// TIA Portal V16 export
// export: Created 2024-12-03T15:41:45.3011474Z, ExportSetting WithReadOnly, DisplayName Totally Integrated Automation Portal, DisplayVersion V16 Update 6, DisplayName TIA Portal Version Control Interface, DisplayVersion V16 Update 2, DisplayName TIA Portal Openness, DisplayVersion V16 Update 6, DisplayName TIA Portal Teamcenter Gateway, DisplayVersion V16, DisplayName SINAMICS Startdrive Advanced, DisplayVersion V16 Update 5, DisplayName SINAMICS Startdrive G130, G150, S120, S150, SINAMICS MV, S210, DisplayVersion V16 Update 5, DisplayName SINAMICS Startdrive G110M, G120, G120C, G120D, G120P, G115D, DisplayVersion V16 Update 5, DisplayName STEP 7 Professional, DisplayVersion V16 Update 6, DisplayName STEP 7 Safety, DisplayVersion V16, DisplayName WinCC Advanced / Unified PC, DisplayVersion V16 Update 6
TYPE "COGNEX_DATAMAN_LOGIC_UDT"
TITLE = SICK Lector/CLV6xx data type
// This data type includes arguments and results using by the SICK_Lector_CLV6xx_PNDP function block.
// stored: CreationDate 2022-02-10T08:20:21.8932261Z, InterfaceModifiedDate 2022-02-10T08:21:18.7143517Z, IsConsistent true, LibraryConformanceStatus The object is library-conformant., ModifiedDate 2022-02-10T08:21:18.7143517Z
   STRUCT
      Cmd : Struct
         Reset : Bool;
         ScanAuto : Bool;
         ScanManual : Bool;
      END_STRUCT;
      Status : Struct
         ReadyForNewScan : Bool;
         ReqDone : Bool;
         ReqBusy : Bool;
         ManualModeActive : Bool;
      END_STRUCT;
      Alarms : Struct
         NotConnected : "HmiAlarm";   // The scanner is not connected
         TimeOutReading : "HmiAlarm";   // Timed out receiving barcode from scanner
         TriggerGuard : "HmiAlarm";   // Trigger received when scanner was parsing previous data
         ErrorFromScanner : "HmiAlarm";   // Error code from scanner
         SerialBufferOverFlow { S7_SetPoint := 'True'} : "HmiAlarm";
         status { S7_SetPoint := 'True'} : Word;
      END_STRUCT;
      DiagNostic : Struct
         GoodReads : UDInt;
         BadReads : UDInt;
         TimeOuts : UDInt;
         MissedTrigger : UDInt;
         OutOfSync : UDInt;
         Scans : UDInt;
         ParsingTime : Time;
      END_STRUCT;
      Settings : Struct
         OnDelay : Time;
         OffDelay : Time;
         TimeOut : Time := t#1s;
      END_STRUCT;
      ReadingResult : Struct
         NewResult_Pulse : Bool;
         GoodRead : Bool;
         BadRead : Bool;
         TimeOut : Bool;
         MissedTrigger : Bool;
         OutOfSync : Bool;
         Barcode : String[136];
         GoodRead_Pulse : Bool;
         BadRead_Pulse : Bool;
         TimeOut_Pulse : Bool;
         MissedTrigger_Pulse : Bool;
         OutOfSync_Pulse : Bool;
         Barcode_Pulse : String[136];
         "Counter" : USInt;   // This counter is incremented if a new reading result has arrived (In)
         Length : Int := 100;   // Byte length of the reading result (Out)
         chars : Array[1..136] of Char;   // Reading result data defined in the SOPAS output format (Out)
      END_STRUCT;
      Tracking : "Tracking_UDT";
      Zone : Int;
      "Name" : String[40];
   END_STRUCT;
END_TYPE
